FUNCTION_BLOCK PUBLIC ABSTRACT FBA_ALARM_HANDLER IMPLEMENTS I_ALARM_HANDLER
VAR_INPUT
END_VAR
VAR_OUTPUT
END_VAR
VAR
END_VAR

METHOD ABSTRACT RegisterAlarm : REFERENCE TO FBA_ALARM_HANDLER
VAR_INPUT
	Alarm	: REFERENCE TO FB_ALARM;
	Prefix	: STRING := '';
	Update : BOOL := TRUE;
END_VAR
END_METHOD

END_FUNCTION_BLOCK

(* stored: Version 1.1.0.1, ProductVersion 3.1.4024.12
   POU FBA_ALARM_HANDLER: Id {28e66e4a-40c9-42c1-ba15-4030d16dee0b}, SpecialFunc None
   Method RegisterAlarm: Id {ea224343-dc7b-4190-8929-085d23df7ce9} *)
